// TIA Portal V19 export
TYPE "LubrPump_Alr"
// stored: Access Published
   STRUCT
      LowLevelLubrication : Bool;
   END_STRUCT;
END_TYPE
